PROGRAM MAIN

(* 
	GOF 		Provide a unified interface to a set of interfaces in a subsystem. 
				Facade defines a higher-level interface that makes the subsystem easier to use.
*)
P_Composite();

END_PROGRAM

(* stored: Version 1.1.0.1, ProductVersion 3.1.4024.12
   POU MAIN: Id {29abbce7-c4e9-4398-9403-4d1c70eab13f}, SpecialFunc None *)
